// TIA Portal V19 export
DATA_BLOCK "GlobalConst_DB"   // DB8
{ S7_Optimized_Access := 'TRUE' }
// stored: MemoryReserve 100
   VAR
      mqtt_host_address : String := '192.168.1.165';
      mqtt_port : UInt := 1883;
      mqtt_username : WString := WSTRING#'mqttbroker';
      mqtt_password : WString := WSTRING#'IoT@2023';
   END_VAR
BEGIN
END_DATA_BLOCK
